TYPE ST_MESSAGE_STATE :
STRUCT
  State         : E_MESSAGE_STATE;  // as always... combined value of Cmd equivalent and e_progress
END_STRUCT
END_TYPE

(* stored: Version 1.1.0.1
   DUT ST_MESSAGE_STATE: Id {33a7da91-0d43-4e0b-90f9-502725f362b7} *)
